INTERFACE I_XplanarTable EXTENDS I_Base, I_DemoStep

PROPERTY Table : I_XPlanarSystem
GET
END_GET
SET
END_SET
END_PROPERTY

END_INTERFACE

(* stored: Version 1.1.0.1, ProductVersion 3.1.4026.20
   Itf I_XplanarTable: Id {393729b2-f9fc-44bd-bd30-109f4eaa1dbd}
   Property Table: Id {9f94cf65-dfe8-4302-a27a-9f5ed784849e}
   Get Get: Id {7991b6d4-1ee7-4fa4-9363-1b0210be66fb}
   Set Set: Id {e67442c7-b59f-4708-8d6e-b5378803d2e4} *)
